TYPE (* logiBUS_DI Struct *)
  (* Version 1.0, 2025-07-21, franz *)
  PACKAGE logiBUS::io::DI_CAN;
  logiBUS_2_CAN_DI_S : STRUCT
    Pin : USINT := 255;
  END_STRUCT;
END_TYPE
